(* Schneider Machine Expert - Basic project Questao4.3_FelipeV1_20241016, file version 2.9.0.0 *)
(* ProjectInformations: Name=Novo projeto *)

HARDWARE
  Cpu 0: TM221M16R/G
  EthernetConfiguration: NetworkName=M221, IpAllocationMode=FixedAddress, IpAddress=0.0.0.0, SubnetMask=0.0.0.0
  SerialLineConfiguration: Baud=Baud19200, Parity=ParityEven, DataBits=DataBits8, StopBits=StopBits1, PhysicalMedium=PhysicalMediumRs485, TransmissionMode=TransmissionModeModbusRtu, SlaveId=1, Addressing=SlaveAddressing
  MastTask: UsePeriodScanMode=false, PeriodScan=100
  FastTask: Period=255
  CpuBehavior: StartingMode=StartAsPreviousState, AutoSaveRamOnEeprom=true, WatchdogPeriod=250

SYMBOLS  (address, symbol, comment, settings)
  %M5       E1_E2_TO_E3
  %M6       E1_E2_TO_E4

GRAFCET Grafcet POU
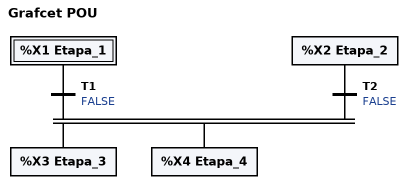
  INITIAL_STEP %X1  (* Etapa_1 *)
  STEP %X2  (* Etapa_2 *)
  STEP %X3  (* Etapa_3 *)
  STEP %X4  (* Etapa_4 *)
  TRANSITION T1 FROM %X1 TO %X3, %X4 := FALSE;
  TRANSITION T2 FROM %X2 TO %X3, %X4 := FALSE;

TRANSITION T1 (%X1 -> %X3, %X4) 
  (* SectionNumber=0 *)

// Rung 0: Tr1
  LD 0
  ENDT
  // as ST:
  //   TRANSITION := FALSE;

TRANSITION T2 (%X2 -> %X3, %X4) 
  (* SectionNumber=0 *)

// Rung 1: Tr2
  LD 0
  ENDT
  // as ST:
  //   TRANSITION := FALSE;

POU Novo POU
  (* SectionNumber=5 *)

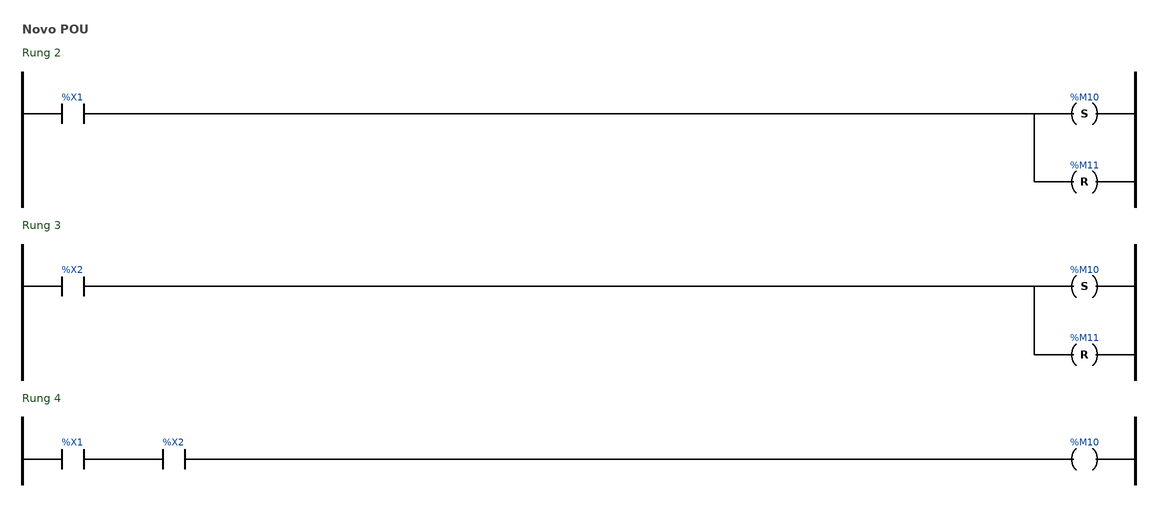

// Rung 2
  LD %X1
  S %M10
  R %M11
  // as ST:
  //   IF %X1 THEN %M10 := TRUE; END_IF;
  //   IF %X1 THEN %M11 := FALSE; END_IF;

// Rung 3
  LD %X2
  S %M10
  R %M11
  // as ST:
  //   IF %X2 THEN %M10 := TRUE; END_IF;
  //   IF %X2 THEN %M11 := FALSE; END_IF;

// Rung 4
  LD %X1
  AND %X2
  ST %M10
  // as ST:
  //   %M10 := %X1 AND %X2;
